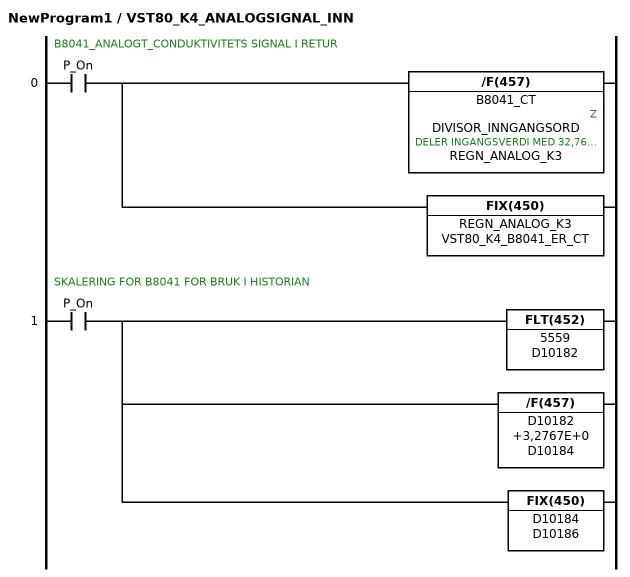
; [picture p480: NewProgram1 / VST80_K4_ANALOGSIGNAL_INN, rungs 0-1]
; rung 0: B8041_ANALOGT_CONDUKTIVITETS SIGNAL I RETUR
LD P_On
/F(457) B8041_CT DIVISOR_INNGANGSORD REGN_ANALOG_K3  ; Z, DELER INGANGSVERDI MED 32,760 FOR OMREGNING TIL 0-1000
FIX(450) REGN_ANALOG_K3 VST80_K4_B8041_ER_CT
; rung 1: SKALERING FOR B8041 FOR BRUK I HISTORIAN
LD P_On
FLT(452) 5559 D10182
/F(457) D10182 +3,2767E+0 D10184
FIX(450) D10184 D10186

### Section VST80_K4_OBJEKTER

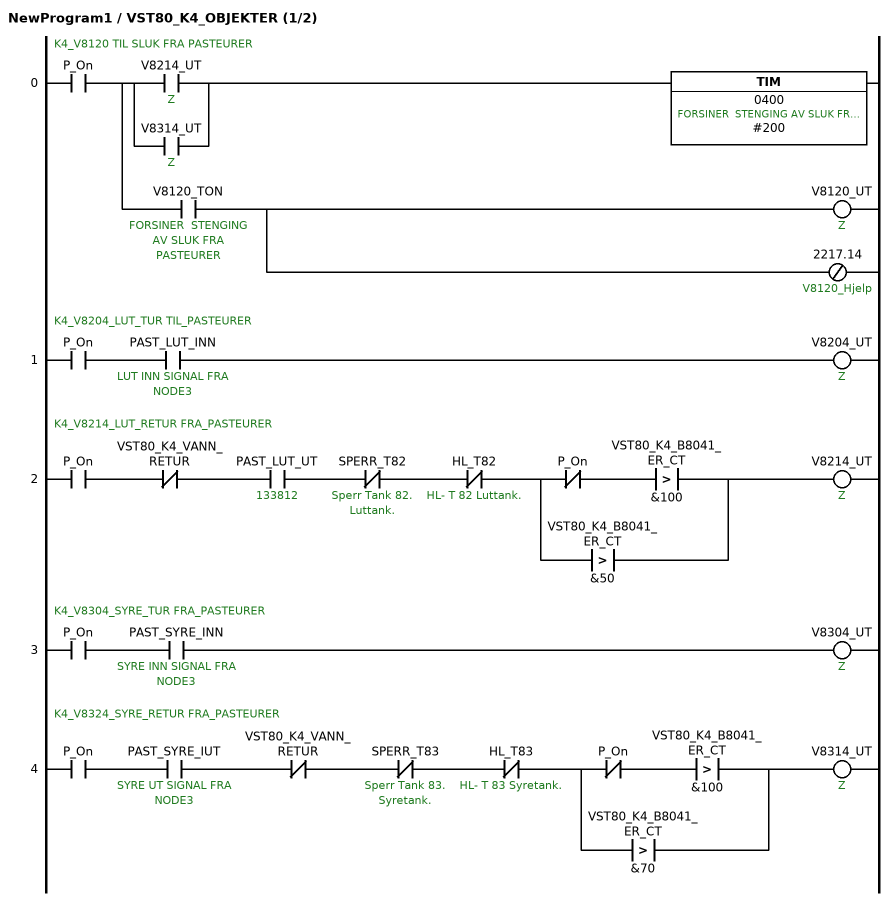
; rung 0: K4_V8120 TIL SLUK FRA PASTEURER
LD P_On
OUT TR0
LD V8214_UT  ; Z
OR V8314_UT  ; Z
ANDLD
TIM 0400 #200  ; FORSINER  STENGING AV SLUK FRA PASTEURER
LD TR0
AND V8120_TON  ; FORSINER  STENGING AV SLUK FRA PASTEURER
OUT V8120_UT  ; Z
OUTNOT 2217.14  ; V8120_Hjelp
; rung 1: K4_V8204_LUT_TUR TIL_PASTEURER
LD P_On
AND PAST_LUT_INN  ; LUT INN SIGNAL FRA NODE3
OUT V8204_UT  ; Z
; rung 2: K4_V8214_LUT_RETUR FRA_PASTEURER
LD P_On
ANDNOT VST80_K4_VANN_RETUR
AND PAST_LUT_UT  ; 133812
ANDNOT SPERR_T82  ; Sperr Tank 82. Luttank.
ANDNOT HL_T82  ; HL- T 82 Luttank.
LDNOT P_On
AND>(320) VST80_K4_B8041_ER_CT &100
OR>(320) VST80_K4_B8041_ER_CT &50
ANDLD
OUT V8214_UT  ; Z
; rung 3: K4_V8304_SYRE_TUR FRA_PASTEURER
LD P_On
AND PAST_SYRE_INN  ; SYRE INN SIGNAL FRA NODE3
OUT V8304_UT  ; Z
; rung 4: K4_V8324_SYRE_RETUR FRA_PASTEURER
LD P_On
AND PAST_SYRE_IUT  ; SYRE UT SIGNAL FRA NODE3
ANDNOT VST80_K4_VANN_RETUR
ANDNOT SPERR_T83  ; Sperr Tank 83. Syretank.
ANDNOT HL_T83  ; HL- T 83 Syretank.
LDNOT P_On
AND>(320) VST80_K4_B8041_ER_CT &100
OR>(320) VST80_K4_B8041_ER_CT &70
ANDLD
OUT V8314_UT  ; Z

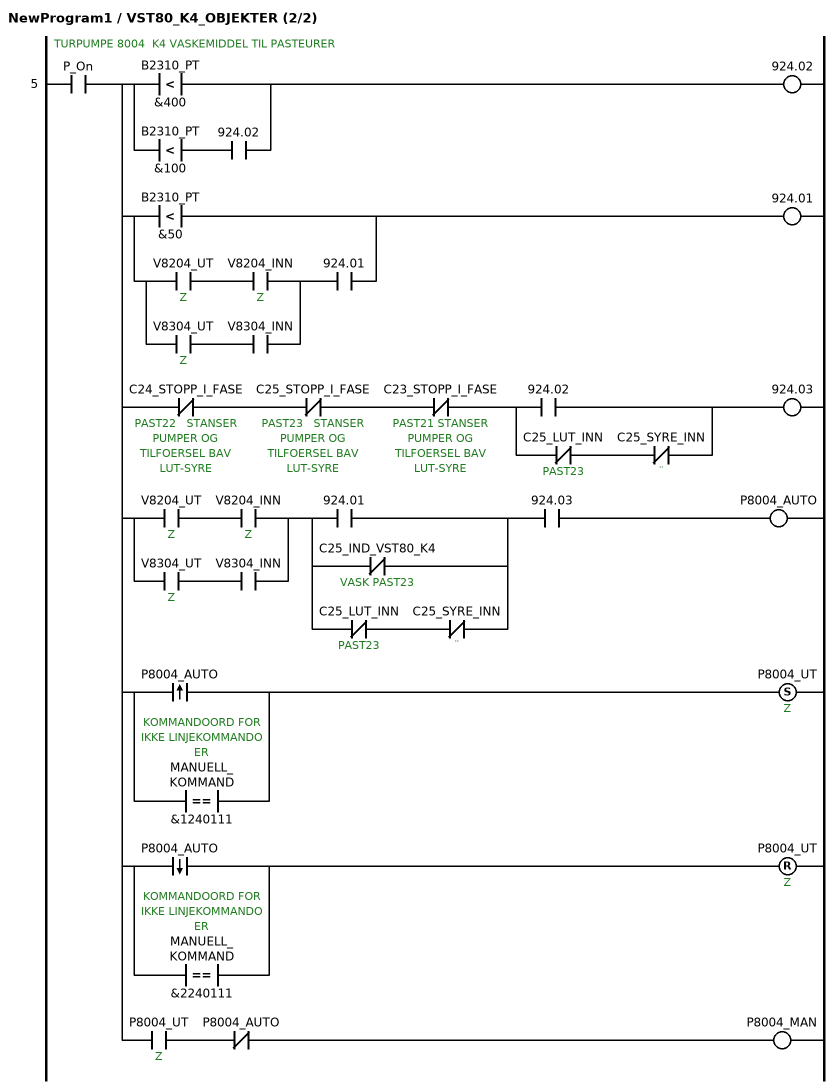
; rung 5: TURPUMPE 8004  K4 VASKEMIDDEL TIL PASTEURER
LD P_On
OUT TR0
LD<(310) B2310_PT &400
LD<(310) B2310_PT &100
AND 924.02
ORLD
ANDLD
OUT 924.02
LD TR0
LD<(310) B2310_PT &50
LD V8204_UT  ; Z
AND V8204_INN  ; Z
LD V8304_UT  ; Z
AND V8304_INN
ORLD
AND 924.01
ORLD
ANDLD
OUT 924.01
LD TR0
ANDNOT C24_STOPP_I_FASE  ; PAST22   STANSER PUMPER OG TILFOERSEL BAV LUT-SYRE
ANDNOT C25_STOPP_I_FASE  ; PAST23   STANSER PUMPER OG TILFOERSEL BAV LUT-SYRE
ANDNOT C23_STOPP_I_FASE  ; PAST21 STANSER PUMPER OG TILFOERSEL BAV LUT-SYRE
LD 924.02
LDNOT C25_LUT_INN  ; PAST23
ANDNOT C25_SYRE_INN  ; ¨
ORLD
ANDLD
OUT 924.03
LD TR0
LD V8204_UT  ; Z
AND V8204_INN  ; Z
LD V8304_UT  ; Z
AND V8304_INN
ORLD
ANDLD
LD 924.01
ORNOT C25_IND_VST80_K4  ; VASK PAST23
LDNOT C25_LUT_INN  ; PAST23
ANDNOT C25_SYRE_INN  ; ¨
ORLD
ANDLD
AND 924.03
OUT P8004_AUTO
LD TR0
@LD P8004_AUTO
OR=L(301) MANUELL_KOMMAND &1240111  ; KOMMANDOORD FOR IKKE LINJEKOMMANDOER
ANDLD
SET P8004_UT  ; Z
LD TR0
%LD P8004_AUTO
OR=L(301) MANUELL_KOMMAND &2240111  ; KOMMANDOORD FOR IKKE LINJEKOMMANDOER
ANDLD
RSET P8004_UT  ; Z
LD TR0
AND P8004_UT  ; Z
ANDNOT P8004_AUTO
OUT P8004_MAN

### Section VST80_FLASH_MOTTAK

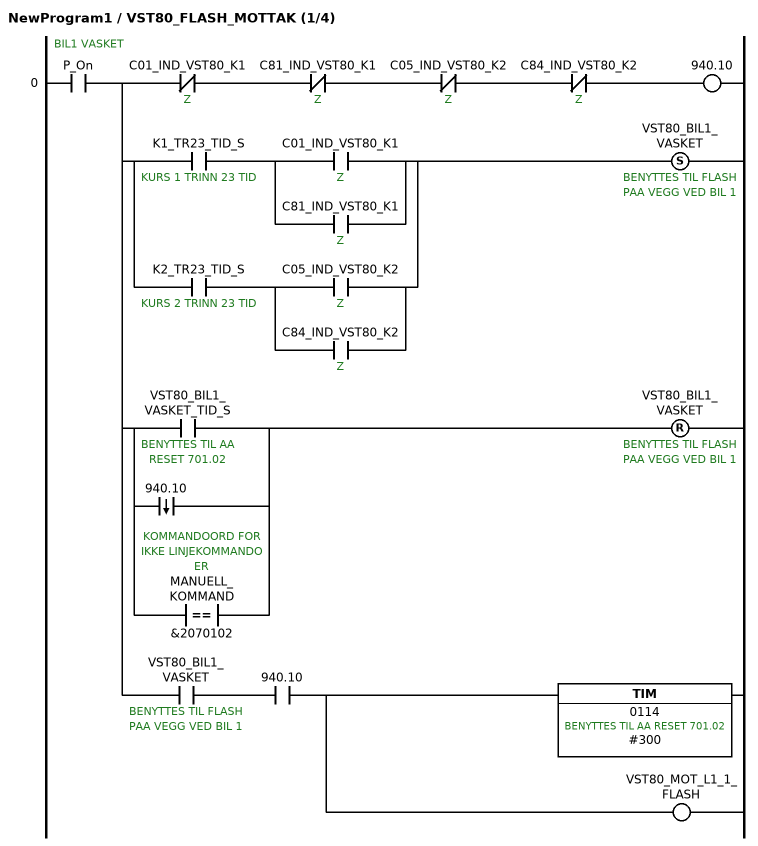
; rung 0: BIL1 VASKET
LD P_On
OUT TR0
ANDNOT C01_IND_VST80_K1  ; Z
ANDNOT C81_IND_VST80_K1  ; Z
ANDNOT C05_IND_VST80_K2  ; Z
ANDNOT C84_IND_VST80_K2  ; Z
OUT 940.10
LD TR0
LD K1_TR23_TID_S  ; KURS 1 TRINN 23 TID
LD C01_IND_VST80_K1  ; Z
OR C81_IND_VST80_K1  ; Z
ANDLD
LD K2_TR23_TID_S  ; KURS 2 TRINN 23 TID
LD C05_IND_VST80_K2  ; Z
OR C84_IND_VST80_K2  ; Z
ANDLD
ORLD
ANDLD
SET VST80_BIL1_VASKET  ; BENYTTES TIL FLASH PAA VEGG VED BIL 1
LD TR0
LD VST80_BIL1_VASKET_TID_S  ; BENYTTES TIL AA RESET 701.02
%OR 940.10
OR=L(301) MANUELL_KOMMAND &2070102  ; KOMMANDOORD FOR IKKE LINJEKOMMANDOER
ANDLD
RSET VST80_BIL1_VASKET  ; BENYTTES TIL FLASH PAA VEGG VED BIL 1
LD TR0
AND VST80_BIL1_VASKET  ; BENYTTES TIL FLASH PAA VEGG VED BIL 1
AND 940.10
TIM 0114 #300  ; BENYTTES TIL AA RESET 701.02
OUT VST80_MOT_L1_1_FLASH

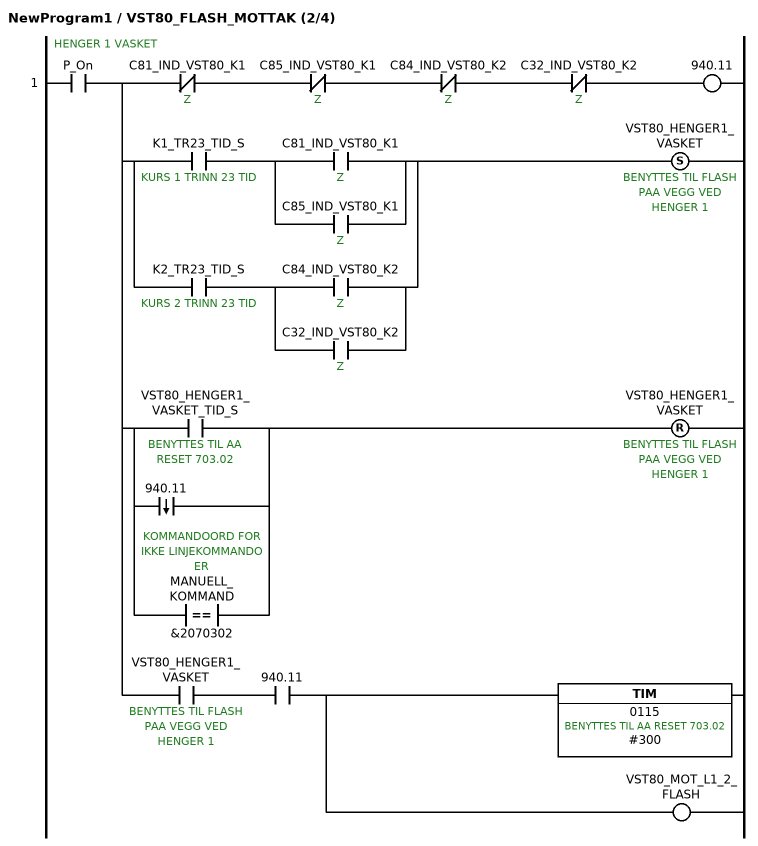
; rung 1: HENGER 1 VASKET
LD P_On
OUT TR0
ANDNOT C81_IND_VST80_K1  ; Z
ANDNOT C85_IND_VST80_K1  ; Z
ANDNOT C84_IND_VST80_K2  ; Z
ANDNOT C32_IND_VST80_K2  ; Z
OUT 940.11
LD TR0
LD K1_TR23_TID_S  ; KURS 1 TRINN 23 TID
LD C81_IND_VST80_K1  ; Z
OR C85_IND_VST80_K1  ; Z
ANDLD
LD K2_TR23_TID_S  ; KURS 2 TRINN 23 TID
LD C84_IND_VST80_K2  ; Z
OR C32_IND_VST80_K2  ; Z
ANDLD
ORLD
ANDLD
SET VST80_HENGER1_VASKET  ; BENYTTES TIL FLASH PAA VEGG VED HENGER 1
LD TR0
LD VST80_HENGER1_VASKET_TID_S  ; BENYTTES TIL AA RESET 703.02
%OR 940.11
OR=L(301) MANUELL_KOMMAND &2070302  ; KOMMANDOORD FOR IKKE LINJEKOMMANDOER
ANDLD
RSET VST80_HENGER1_VASKET  ; BENYTTES TIL FLASH PAA VEGG VED HENGER 1
LD TR0
AND VST80_HENGER1_VASKET  ; BENYTTES TIL FLASH PAA VEGG VED HENGER 1
AND 940.11
TIM 0115 #300  ; BENYTTES TIL AA RESET 703.02
OUT VST80_MOT_L1_2_FLASH

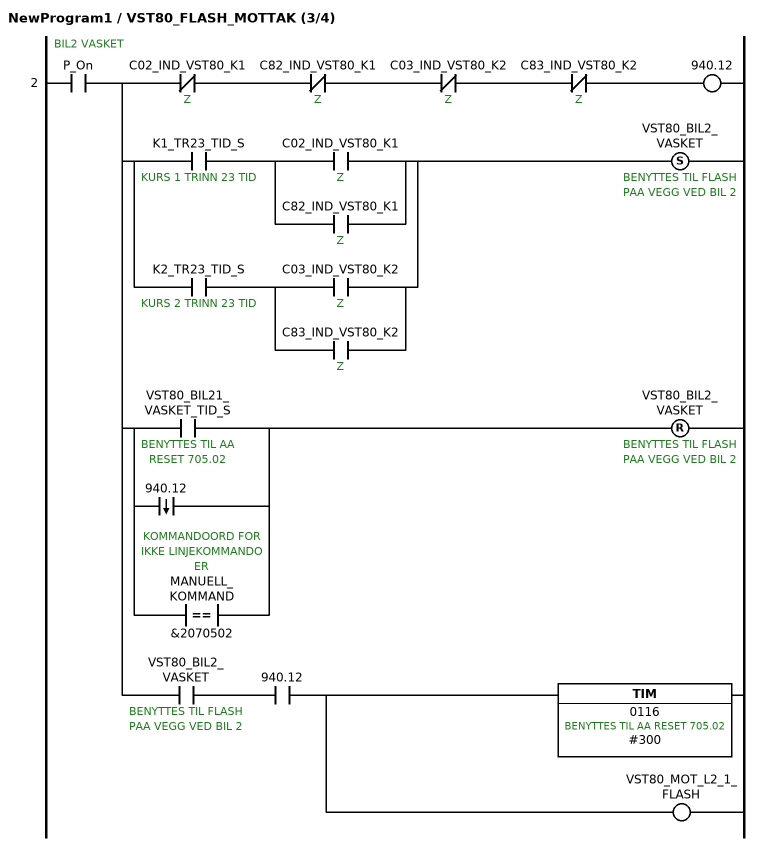
; rung 2: BIL2 VASKET
LD P_On
OUT TR0
ANDNOT C02_IND_VST80_K1  ; Z
ANDNOT C82_IND_VST80_K1  ; Z
ANDNOT C03_IND_VST80_K2  ; Z
ANDNOT C83_IND_VST80_K2  ; Z
OUT 940.12
LD TR0
LD K1_TR23_TID_S  ; KURS 1 TRINN 23 TID
LD C02_IND_VST80_K1  ; Z
OR C82_IND_VST80_K1  ; Z
ANDLD
LD K2_TR23_TID_S  ; KURS 2 TRINN 23 TID
LD C03_IND_VST80_K2  ; Z
OR C83_IND_VST80_K2  ; Z
ANDLD
ORLD
ANDLD
SET VST80_BIL2_VASKET  ; BENYTTES TIL FLASH PAA VEGG VED BIL 2
LD TR0
LD VST80_BIL21_VASKET_TID_S  ; BENYTTES TIL AA RESET 705.02
%OR 940.12
OR=L(301) MANUELL_KOMMAND &2070502  ; KOMMANDOORD FOR IKKE LINJEKOMMANDOER
ANDLD
RSET VST80_BIL2_VASKET  ; BENYTTES TIL FLASH PAA VEGG VED BIL 2
LD TR0
AND VST80_BIL2_VASKET  ; BENYTTES TIL FLASH PAA VEGG VED BIL 2
AND 940.12
TIM 0116 #300  ; BENYTTES TIL AA RESET 705.02
OUT VST80_MOT_L2_1_FLASH

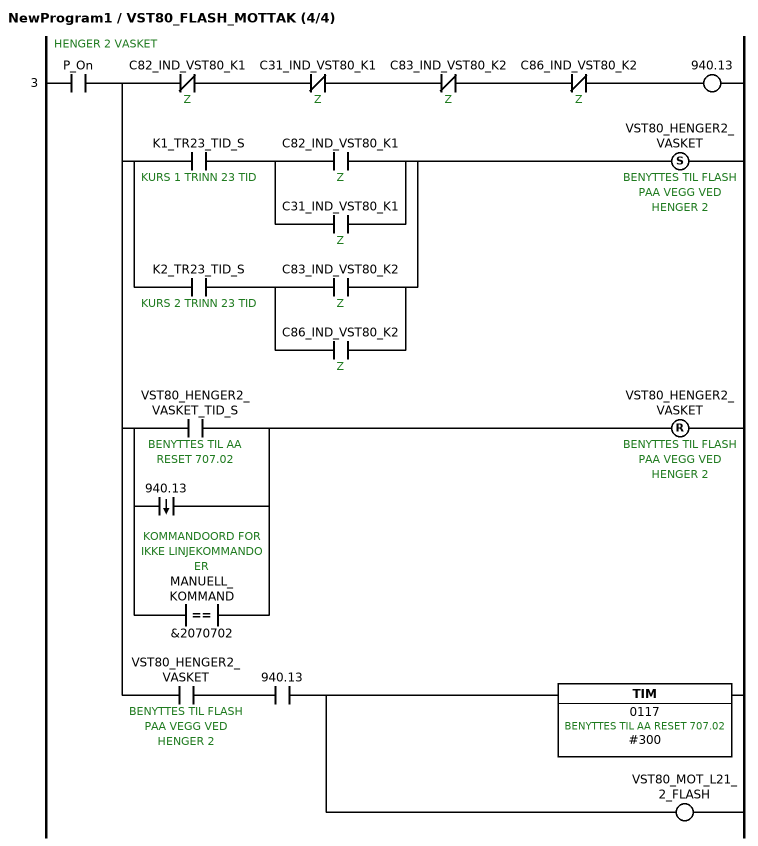
; rung 3: HENGER 2 VASKET
LD P_On
OUT TR0
ANDNOT C82_IND_VST80_K1  ; Z
ANDNOT C31_IND_VST80_K1  ; Z
ANDNOT C83_IND_VST80_K2  ; Z
ANDNOT C86_IND_VST80_K2  ; Z
OUT 940.13
LD TR0
LD K1_TR23_TID_S  ; KURS 1 TRINN 23 TID
LD C82_IND_VST80_K1  ; Z
OR C31_IND_VST80_K1  ; Z
ANDLD
LD K2_TR23_TID_S  ; KURS 2 TRINN 23 TID
LD C83_IND_VST80_K2  ; Z
OR C86_IND_VST80_K2  ; Z
ANDLD
ORLD
ANDLD
SET VST80_HENGER2_VASKET  ; BENYTTES TIL FLASH PAA VEGG VED HENGER 2
LD TR0
LD VST80_HENGER2_VASKET_TID_S  ; BENYTTES TIL AA RESET 707.02
%OR 940.13
OR=L(301) MANUELL_KOMMAND &2070702  ; KOMMANDOORD FOR IKKE LINJEKOMMANDOER
ANDLD
RSET VST80_HENGER2_VASKET  ; BENYTTES TIL FLASH PAA VEGG VED HENGER 2
LD TR0
AND VST80_HENGER2_VASKET  ; BENYTTES TIL FLASH PAA VEGG VED HENGER 2
AND 940.13
TIM 0117 #300  ; BENYTTES TIL AA RESET 707.02
OUT VST80_MOT_L21_2_FLASH

### Section PGM_500_VST80_KURS1

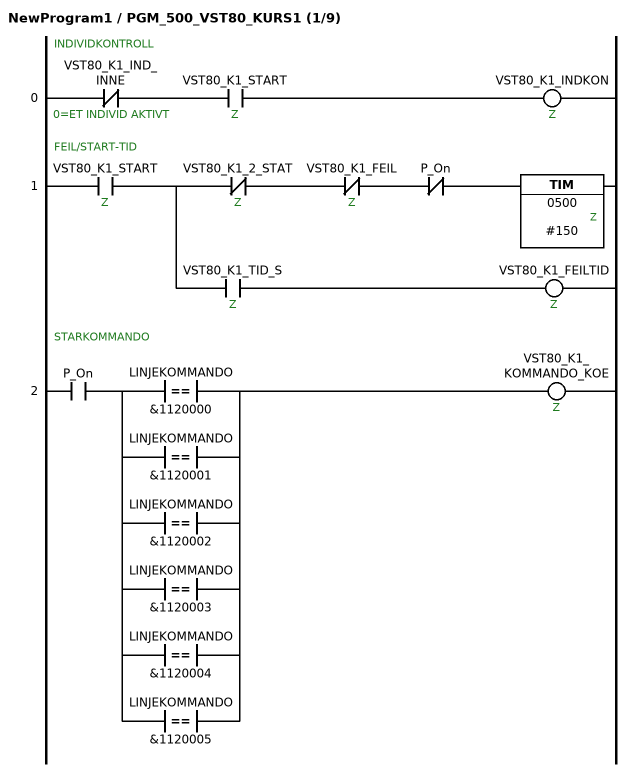
; rung 0: INDIVIDKONTROLL
LDNOT VST80_K1_IND_INNE  ; 0=ET INDIVID AKTIVT
AND VST80_K1_START  ; Z
OUT VST80_K1_INDKON  ; Z
; rung 1: FEIL/START-TID
LD VST80_K1_START  ; Z
OUT TR0
ANDNOT VST80_K1_2_STAT  ; Z
ANDNOT VST80_K1_FEIL  ; Z
ANDNOT P_On
TIM 0500 #150  ; Z
LD TR0
AND VST80_K1_TID_S  ; Z
OUT VST80_K1_FEILTID  ; Z
; rung 2: STARKOMMANDO
LD P_On
LD=L(301) LINJEKOMMANDO &1120000
OR=L(301) LINJEKOMMANDO &1120001
OR=L(301) LINJEKOMMANDO &1120002
OR=L(301) LINJEKOMMANDO &1120003
OR=L(301) LINJEKOMMANDO &1120004
OR=L(301) LINJEKOMMANDO &1120005
ANDLD
OUT VST80_K1_KOMMANDO_KOE  ; Z

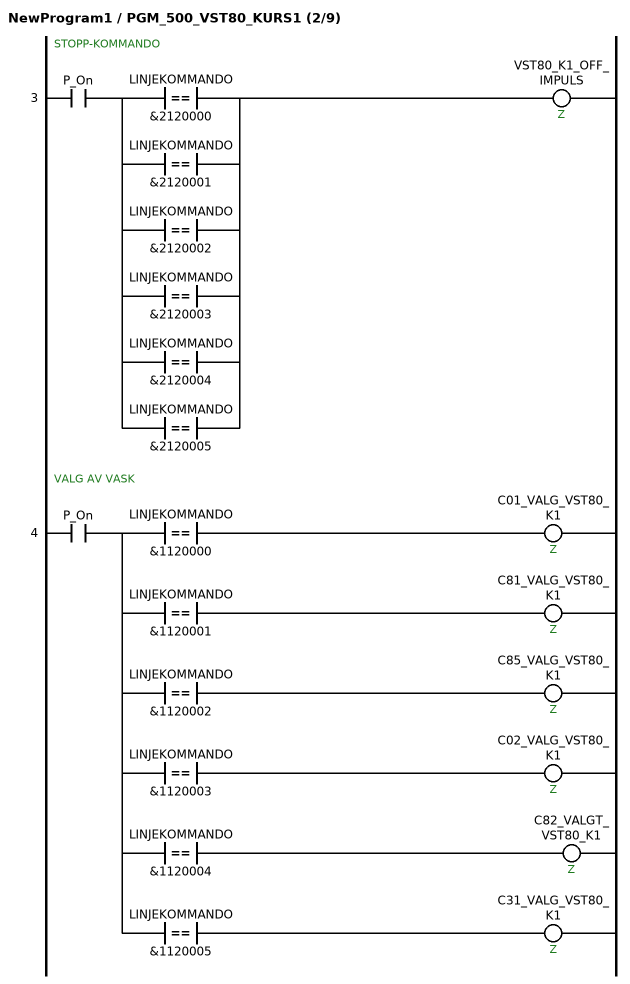
; rung 3: STOPP-KOMMANDO
LD P_On
LD=L(301) LINJEKOMMANDO &2120000
OR=L(301) LINJEKOMMANDO &2120001
OR=L(301) LINJEKOMMANDO &2120002
OR=L(301) LINJEKOMMANDO &2120003
OR=L(301) LINJEKOMMANDO &2120004
OR=L(301) LINJEKOMMANDO &2120005
ANDLD
OUT VST80_K1_OFF_IMPULS  ; Z
; rung 4: VALG AV VASK
LD P_On
OUT TR0
AND=L(301) LINJEKOMMANDO &1120000
OUT C01_VALG_VST80_K1  ; Z
LD TR0
AND=L(301) LINJEKOMMANDO &1120001
OUT C81_VALG_VST80_K1  ; Z
LD TR0
AND=L(301) LINJEKOMMANDO &1120002
OUT C85_VALG_VST80_K1  ; Z
LD TR0
AND=L(301) LINJEKOMMANDO &1120003
OUT C02_VALG_VST80_K1  ; Z
LD TR0
AND=L(301) LINJEKOMMANDO &1120004
OUT C82_VALGT_VST80_K1  ; Z
LD TR0
AND=L(301) LINJEKOMMANDO &1120005
OUT C31_VALG_VST80_K1  ; Z

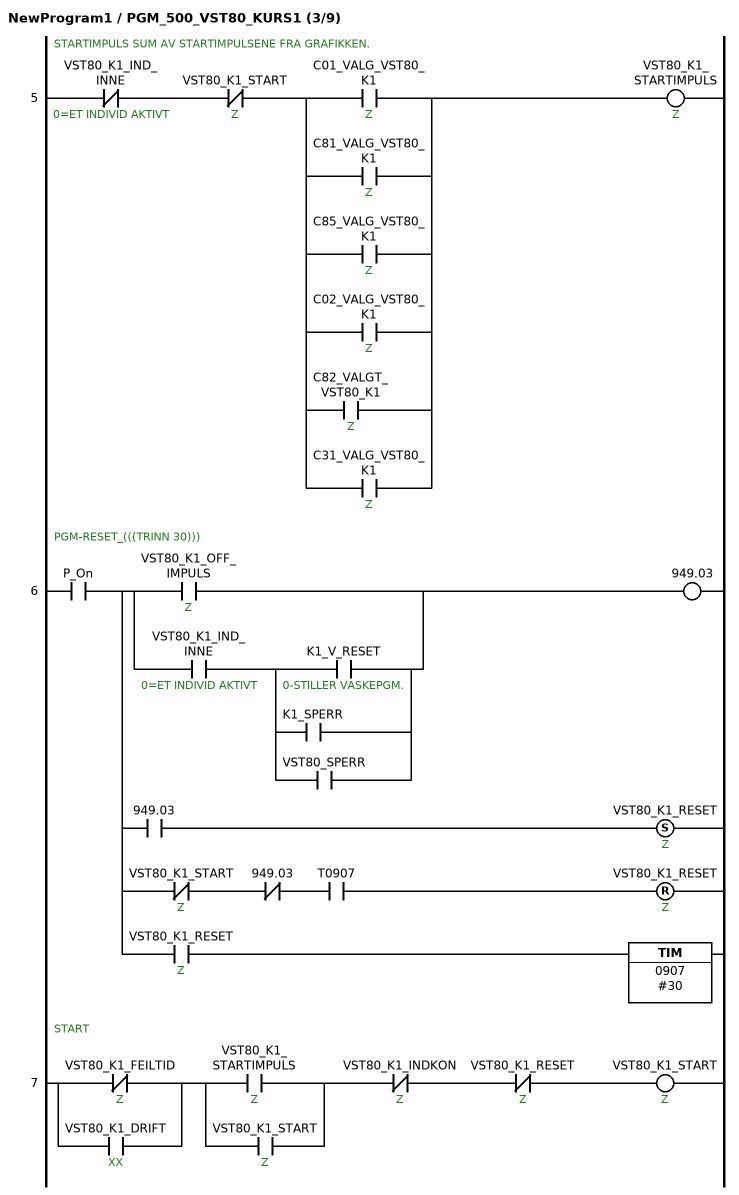
; rung 5: STARTIMPULS SUM AV STARTIMPULSENE FRA GRAFIKKEN.
LDNOT VST80_K1_IND_INNE  ; 0=ET INDIVID AKTIVT
ANDNOT VST80_K1_START  ; Z
LD C01_VALG_VST80_K1  ; Z
OR C81_VALG_VST80_K1  ; Z
OR C85_VALG_VST80_K1  ; Z
OR C02_VALG_VST80_K1  ; Z
OR C82_VALGT_VST80_K1  ; Z
OR C31_VALG_VST80_K1  ; Z
ANDLD
OUT VST80_K1_STARTIMPULS  ; Z
; rung 6: PGM-RESET_(((TRINN 30)))
LD P_On
OUT TR0
LD VST80_K1_OFF_IMPULS  ; Z
LD VST80_K1_IND_INNE  ; 0=ET INDIVID AKTIVT
LD K1_V_RESET  ; 0-STILLER VASKEPGM.
OR K1_SPERR
OR VST80_SPERR
ANDLD
ORLD
ANDLD
OUT 949.03
LD TR0
AND 949.03
SET VST80_K1_RESET  ; Z
LD TR0
ANDNOT VST80_K1_START  ; Z
ANDNOT 949.03
AND T0907
RSET VST80_K1_RESET  ; Z
LD TR0
AND VST80_K1_RESET  ; Z
TIM 0907 #30
; rung 7: START
LDNOT VST80_K1_FEILTID  ; Z
OR VST80_K1_DRIFT  ; XX
LD VST80_K1_STARTIMPULS  ; Z
OR VST80_K1_START  ; Z
ANDLD
ANDNOT VST80_K1_INDKON  ; Z
ANDNOT VST80_K1_RESET  ; Z
OUT VST80_K1_START  ; Z

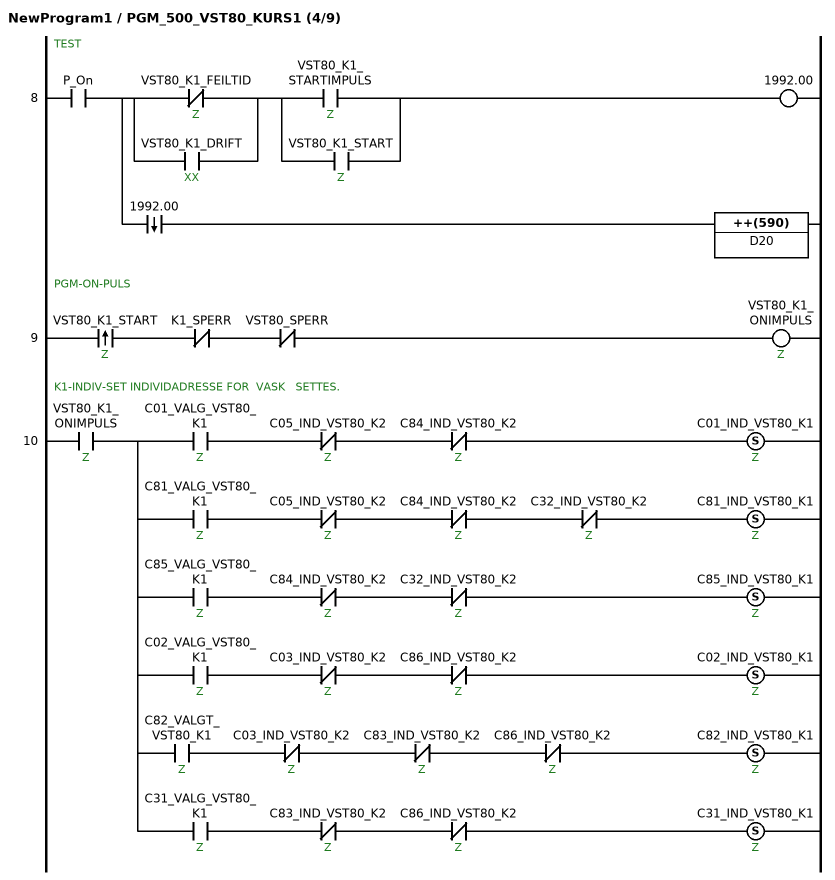
; rung 8: TEST
LD P_On
OUT TR0
LDNOT VST80_K1_FEILTID  ; Z
OR VST80_K1_DRIFT  ; XX
ANDLD
LD VST80_K1_STARTIMPULS  ; Z
OR VST80_K1_START  ; Z
ANDLD
OUT 1992.00
LD TR0
%AND 1992.00
++(590) D20
; rung 9: PGM-ON-PULS
@LD VST80_K1_START  ; Z
ANDNOT K1_SPERR
ANDNOT VST80_SPERR
OUT VST80_K1_ONIMPULS  ; Z
; rung 10: K1-INDIV-SET INDIVIDADRESSE FOR  VASK   SETTES.
LD VST80_K1_ONIMPULS  ; Z
OUT TR0
AND C01_VALG_VST80_K1  ; Z
ANDNOT C05_IND_VST80_K2  ; Z
ANDNOT C84_IND_VST80_K2  ; Z
SET C01_IND_VST80_K1  ; Z
LD TR0
AND C81_VALG_VST80_K1  ; Z
ANDNOT C05_IND_VST80_K2  ; Z
ANDNOT C84_IND_VST80_K2  ; Z
ANDNOT C32_IND_VST80_K2  ; Z
SET C81_IND_VST80_K1  ; Z
LD TR0
AND C85_VALG_VST80_K1  ; Z
ANDNOT C84_IND_VST80_K2  ; Z
ANDNOT C32_IND_VST80_K2  ; Z
SET C85_IND_VST80_K1  ; Z
LD TR0
AND C02_VALG_VST80_K1  ; Z
ANDNOT C03_IND_VST80_K2  ; Z
ANDNOT C86_IND_VST80_K2  ; Z
SET C02_IND_VST80_K1  ; Z
LD TR0
AND C82_VALGT_VST80_K1  ; Z
ANDNOT C03_IND_VST80_K2  ; Z
ANDNOT C83_IND_VST80_K2  ; Z
ANDNOT C86_IND_VST80_K2  ; Z
SET C82_IND_VST80_K1  ; Z
LD TR0
AND C31_VALG_VST80_K1  ; Z
ANDNOT C83_IND_VST80_K2  ; Z
ANDNOT C86_IND_VST80_K2  ; Z
SET C31_IND_VST80_K1  ; Z

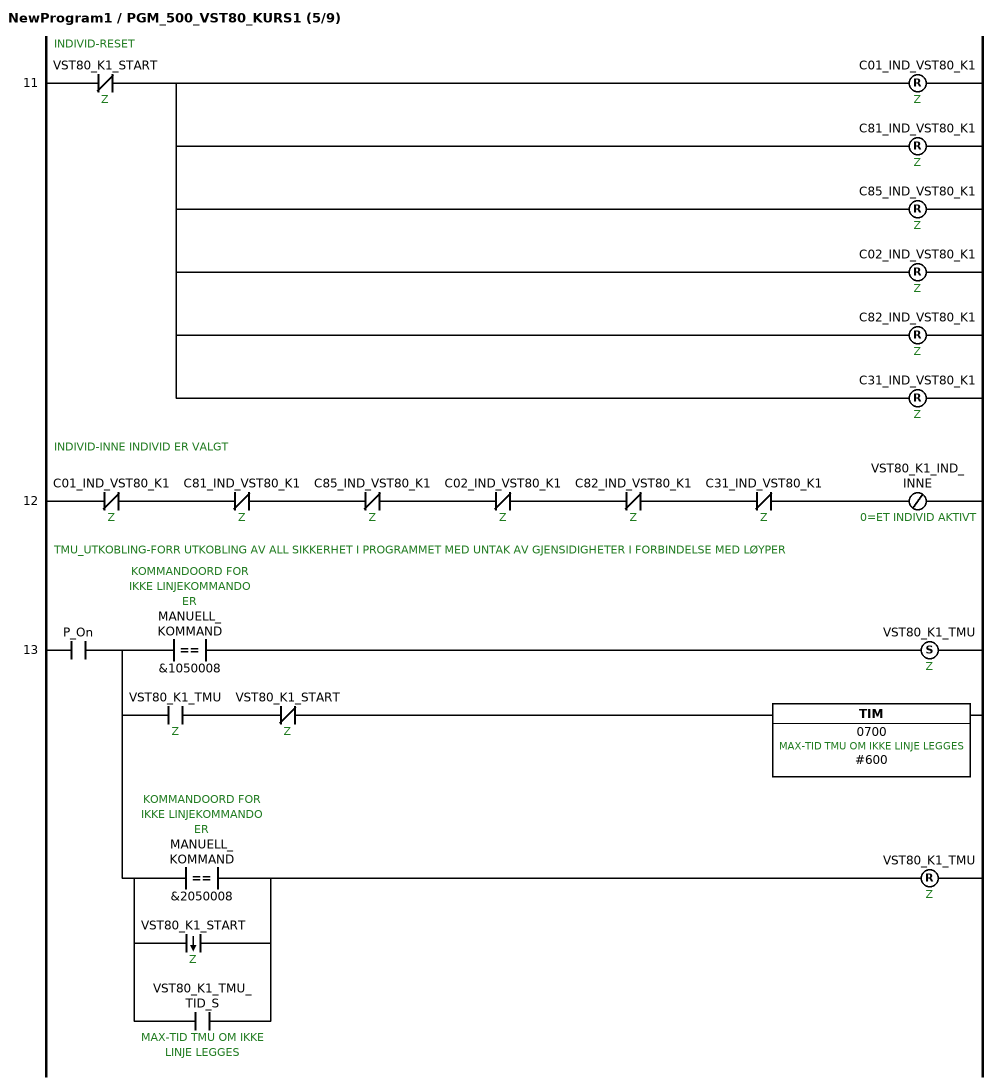
; rung 11: INDIVID-RESET
LDNOT VST80_K1_START  ; Z
RSET C01_IND_VST80_K1  ; Z
RSET C81_IND_VST80_K1  ; Z
RSET C85_IND_VST80_K1  ; Z
RSET C02_IND_VST80_K1  ; Z
RSET C82_IND_VST80_K1  ; Z
RSET C31_IND_VST80_K1  ; Z
; rung 12: INDIVID-INNE INDIVID ER VALGT
LDNOT C01_IND_VST80_K1  ; Z
ANDNOT C81_IND_VST80_K1  ; Z
ANDNOT C85_IND_VST80_K1  ; Z
ANDNOT C02_IND_VST80_K1  ; Z
ANDNOT C82_IND_VST80_K1  ; Z
ANDNOT C31_IND_VST80_K1  ; Z
OUTNOT VST80_K1_IND_INNE  ; 0=ET INDIVID AKTIVT
; rung 13: TMU_UTKOBLING-FORR UTKOBLING AV ALL SIKKERHET I PROGRAMMET MED UNTAK AV GJENSIDIGHETER I FORBINDELSE MED LØYPER
LD P_On
OUT TR0
AND=L(301) MANUELL_KOMMAND &1050008  ; KOMMANDOORD FOR IKKE LINJEKOMMANDOER
SET VST80_K1_TMU  ; Z
LD TR0
AND VST80_K1_TMU  ; Z
ANDNOT VST80_K1_START  ; Z
TIM 0700 #600  ; MAX-TID TMU OM IKKE LINJE LEGGES
LD TR0
LD=L(301) MANUELL_KOMMAND &2050008  ; KOMMANDOORD FOR IKKE LINJEKOMMANDOER
%OR VST80_K1_START  ; Z
OR VST80_K1_TMU_TID_S  ; MAX-TID TMU OM IKKE LINJE LEGGES
ANDLD
RSET VST80_K1_TMU  ; Z

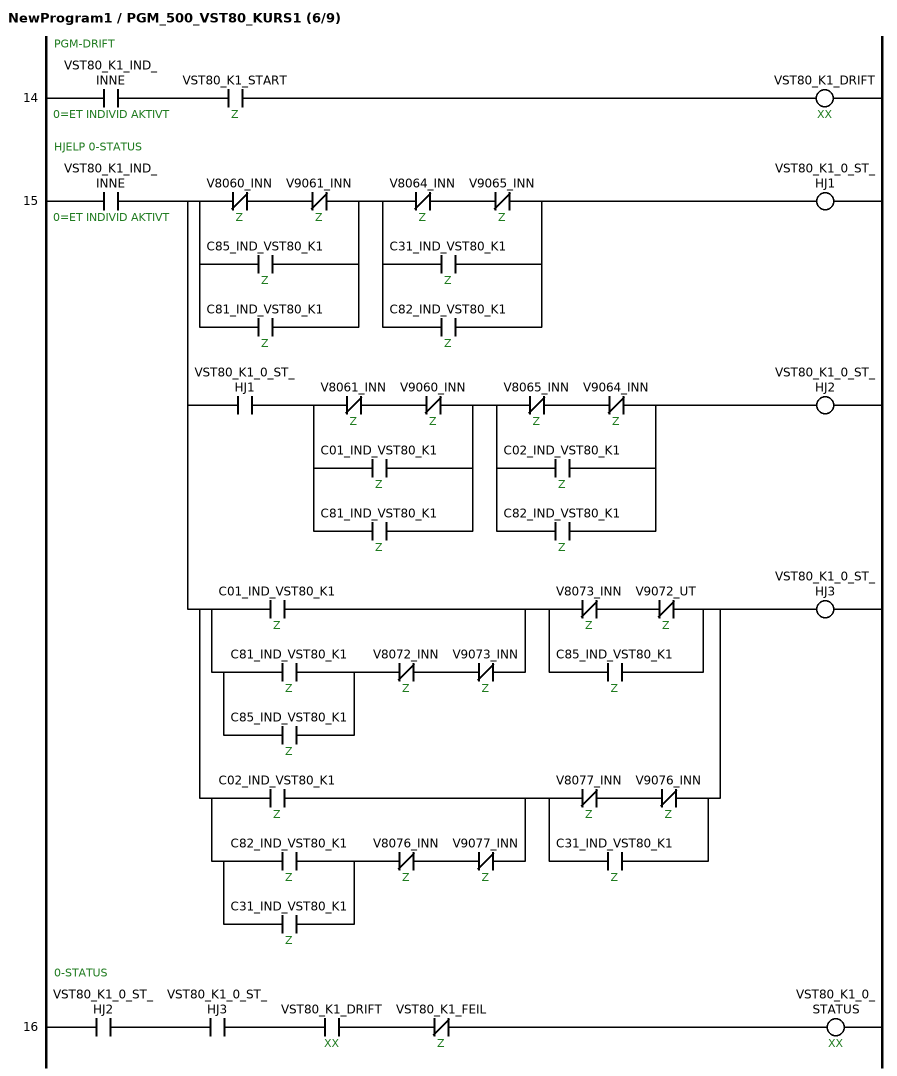
; rung 14: PGM-DRIFT
LD VST80_K1_IND_INNE  ; 0=ET INDIVID AKTIVT
AND VST80_K1_START  ; Z
OUT VST80_K1_DRIFT  ; XX
; rung 15: HJELP 0-STATUS
LD VST80_K1_IND_INNE  ; 0=ET INDIVID AKTIVT
OUT TR0
LDNOT V8060_INN  ; Z
ANDNOT V9061_INN  ; Z
OR C85_IND_VST80_K1  ; Z
OR C81_IND_VST80_K1  ; Z
ANDLD
LDNOT V8064_INN  ; Z
ANDNOT V9065_INN  ; Z
OR C31_IND_VST80_K1  ; Z
OR C82_IND_VST80_K1  ; Z
ANDLD
OUT VST80_K1_0_ST_HJ1
LD TR0
AND VST80_K1_0_ST_HJ1
LDNOT V8061_INN  ; Z
ANDNOT V9060_INN  ; Z
OR C01_IND_VST80_K1  ; Z
OR C81_IND_VST80_K1  ; Z
ANDLD
LDNOT V8065_INN  ; Z
ANDNOT V9064_INN  ; Z
OR C02_IND_VST80_K1  ; Z
OR C82_IND_VST80_K1  ; Z
ANDLD
OUT VST80_K1_0_ST_HJ2
LD TR0
LD C01_IND_VST80_K1  ; Z
LD C81_IND_VST80_K1  ; Z
OR C85_IND_VST80_K1  ; Z
ANDNOT V8072_INN  ; Z
ANDNOT V9073_INN  ; Z
ORLD
LDNOT V8073_INN  ; Z
ANDNOT V9072_UT  ; Z
OR C85_IND_VST80_K1  ; Z
ANDLD
LD C02_IND_VST80_K1  ; Z
LD C82_IND_VST80_K1  ; Z
OR C31_IND_VST80_K1  ; Z
ANDNOT V8076_INN  ; Z
ANDNOT V9077_INN  ; Z
ORLD
LDNOT V8077_INN  ; Z
ANDNOT V9076_INN  ; Z
OR C31_IND_VST80_K1  ; Z
ANDLD
ORLD
ANDLD
OUT VST80_K1_0_ST_HJ3
; rung 16: 0-STATUS
LD VST80_K1_0_ST_HJ2
AND VST80_K1_0_ST_HJ3
AND VST80_K1_DRIFT  ; XX
ANDNOT VST80_K1_FEIL  ; Z
OUT VST80_K1_0_STATUS  ; XX

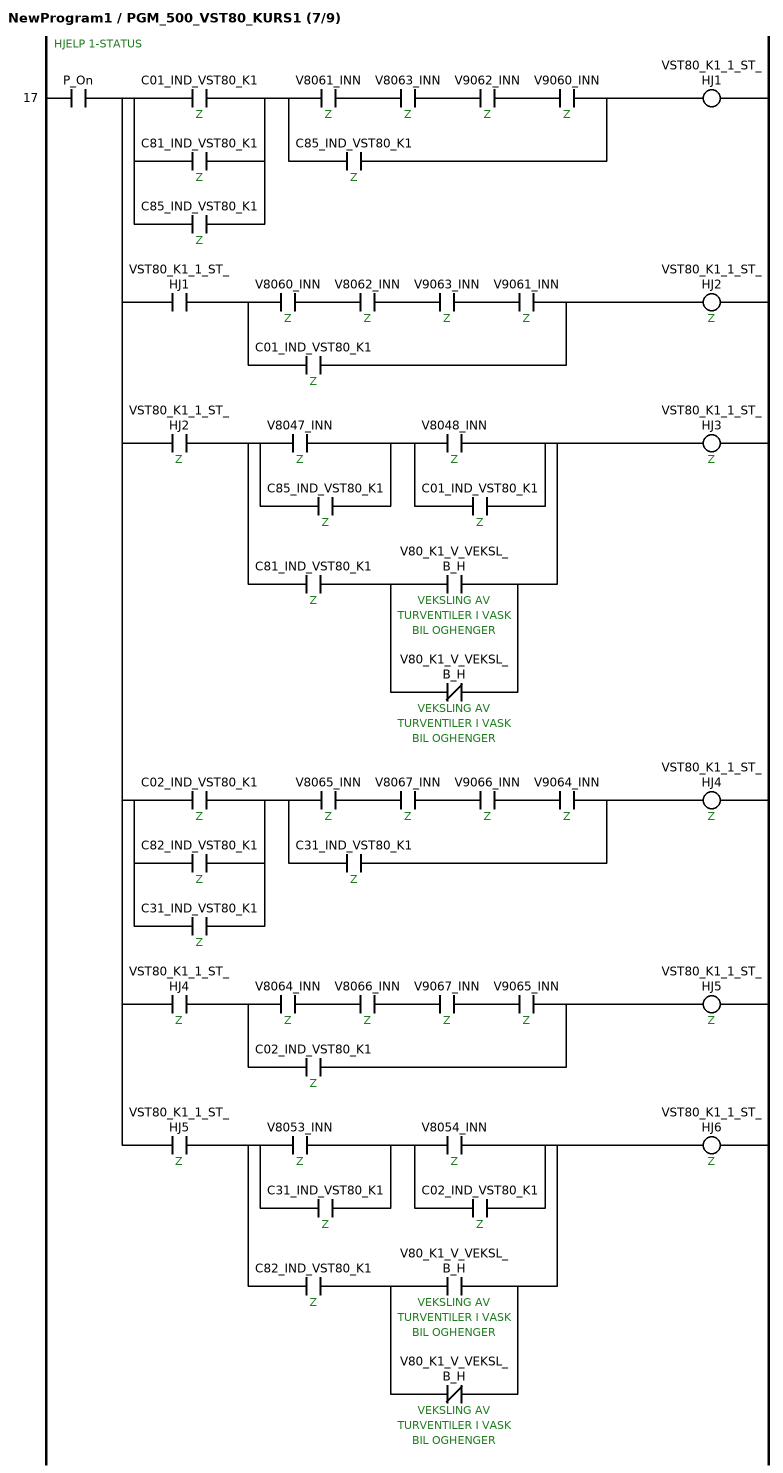
; rung 17: HJELP 1-STATUS
LD P_On
OUT TR0
LD C01_IND_VST80_K1  ; Z
OR C81_IND_VST80_K1  ; Z
OR C85_IND_VST80_K1  ; Z
ANDLD
LD V8061_INN  ; Z
AND V8063_INN  ; Z
AND V9062_INN  ; Z
AND V9060_INN  ; Z
OR C85_IND_VST80_K1  ; Z
ANDLD
OUT VST80_K1_1_ST_HJ1
LD TR0
AND VST80_K1_1_ST_HJ1
LD V8060_INN  ; Z
AND V8062_INN  ; Z
AND V9063_INN  ; Z
AND V9061_INN  ; Z
OR C01_IND_VST80_K1  ; Z
ANDLD
OUT VST80_K1_1_ST_HJ2  ; Z
LD TR0
AND VST80_K1_1_ST_HJ2  ; Z
LD V8047_INN  ; Z
OR C85_IND_VST80_K1  ; Z
LD V8048_INN  ; Z
OR C01_IND_VST80_K1  ; Z
ANDLD
LD C81_IND_VST80_K1  ; Z
LD V80_K1_V_VEKSL_B_H  ; VEKSLING AV TURVENTILER I VASK BIL OGHENGER
ORNOT V80_K1_V_VEKSL_B_H  ; VEKSLING AV TURVENTILER I VASK BIL OGHENGER
ANDLD
ORLD
ANDLD
OUT VST80_K1_1_ST_HJ3  ; Z
LD TR0
LD C02_IND_VST80_K1  ; Z
OR C82_IND_VST80_K1  ; Z
OR C31_IND_VST80_K1  ; Z
ANDLD
LD V8065_INN  ; Z
AND V8067_INN  ; Z
AND V9066_INN  ; Z
AND V9064_INN  ; Z
OR C31_IND_VST80_K1  ; Z
ANDLD
OUT VST80_K1_1_ST_HJ4  ; Z
LD TR0
AND VST80_K1_1_ST_HJ4  ; Z
LD V8064_INN  ; Z
AND V8066_INN  ; Z
AND V9067_INN  ; Z
AND V9065_INN  ; Z
OR C02_IND_VST80_K1  ; Z
ANDLD
OUT VST80_K1_1_ST_HJ5  ; Z
LD TR0
AND VST80_K1_1_ST_HJ5  ; Z
LD V8053_INN  ; Z
OR C31_IND_VST80_K1  ; Z
LD V8054_INN  ; Z
OR C02_IND_VST80_K1  ; Z
ANDLD
LD C82_IND_VST80_K1  ; Z
LD V80_K1_V_VEKSL_B_H  ; VEKSLING AV TURVENTILER I VASK BIL OGHENGER
ORNOT V80_K1_V_VEKSL_B_H  ; VEKSLING AV TURVENTILER I VASK BIL OGHENGER
ANDLD
ORLD
ANDLD
OUT VST80_K1_1_ST_HJ6  ; Z

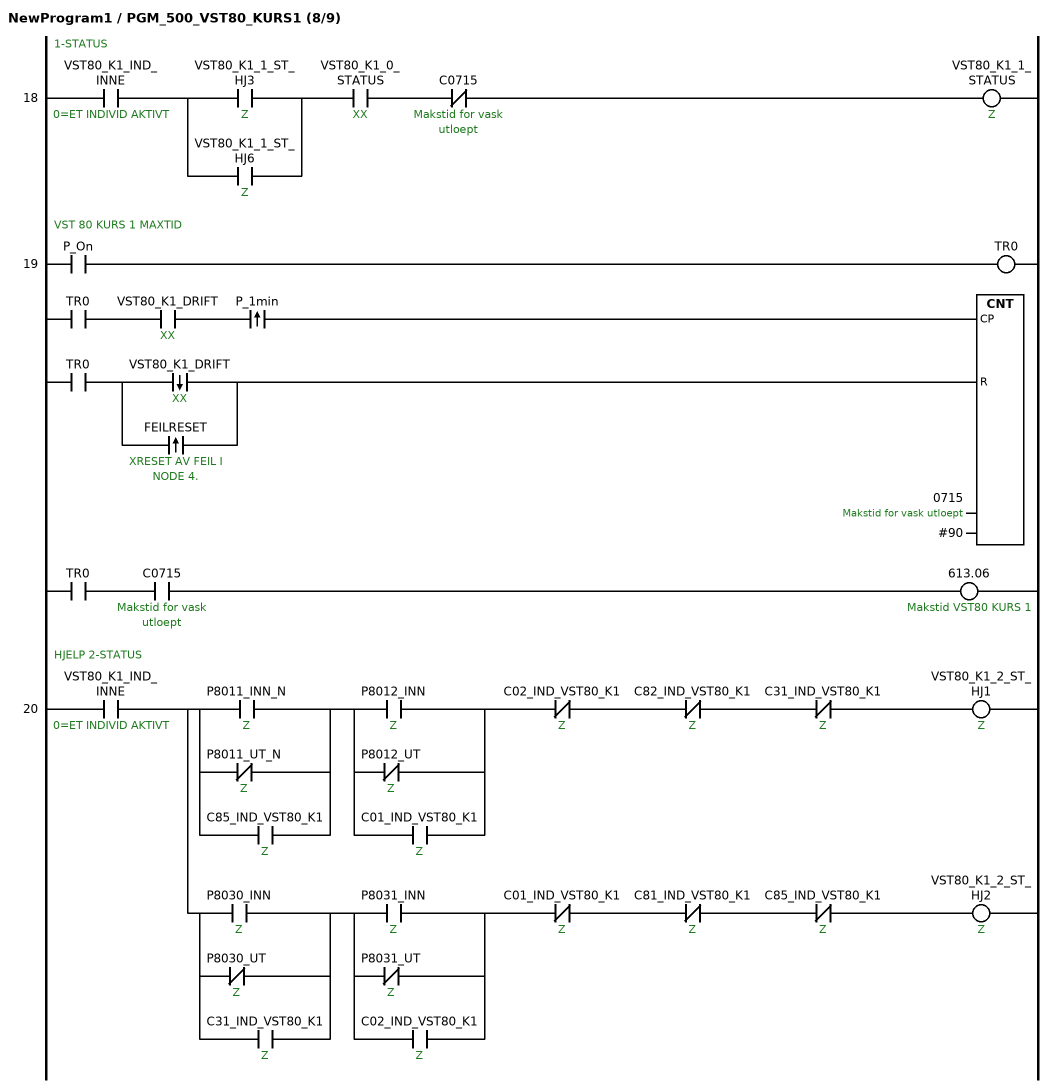
; rung 18: 1-STATUS
LD VST80_K1_IND_INNE  ; 0=ET INDIVID AKTIVT
LD VST80_K1_1_ST_HJ3  ; Z
OR VST80_K1_1_ST_HJ6  ; Z
ANDLD
AND VST80_K1_0_STATUS  ; XX
ANDNOT C0715  ; Makstid for vask utloept
OUT VST80_K1_1_STATUS  ; Z
; rung 19: VST 80 KURS 1 MAXTID
LD P_On
OUT TR0
AND VST80_K1_DRIFT  ; XX
@AND P_1min
LD TR0
%LD VST80_K1_DRIFT  ; XX
@OR FEILRESET  ; XRESET AV FEIL I NODE 4.
ANDLD
CNT 0715 #90  ; Makstid for vask utloept
LD TR0
AND C0715  ; Makstid for vask utloept
OUT 613.06  ; Makstid VST80 KURS 1
; rung 20: HJELP 2-STATUS
LD VST80_K1_IND_INNE  ; 0=ET INDIVID AKTIVT
OUT TR0
LD P8011_INN_N  ; Z
ORNOT P8011_UT_N  ; Z
OR C85_IND_VST80_K1  ; Z
ANDLD
LD P8012_INN  ; Z
ORNOT P8012_UT  ; Z
OR C01_IND_VST80_K1  ; Z
ANDLD
ANDNOT C02_IND_VST80_K1  ; Z
ANDNOT C82_IND_VST80_K1  ; Z
ANDNOT C31_IND_VST80_K1  ; Z
OUT VST80_K1_2_ST_HJ1  ; Z
LD TR0
LD P8030_INN  ; Z
ORNOT P8030_UT  ; Z
OR C31_IND_VST80_K1  ; Z
ANDLD
LD P8031_INN  ; Z
ORNOT P8031_UT  ; Z
OR C02_IND_VST80_K1  ; Z
ANDLD
ANDNOT C01_IND_VST80_K1  ; Z
ANDNOT C81_IND_VST80_K1  ; Z
ANDNOT C85_IND_VST80_K1  ; Z
OUT VST80_K1_2_ST_HJ2  ; Z

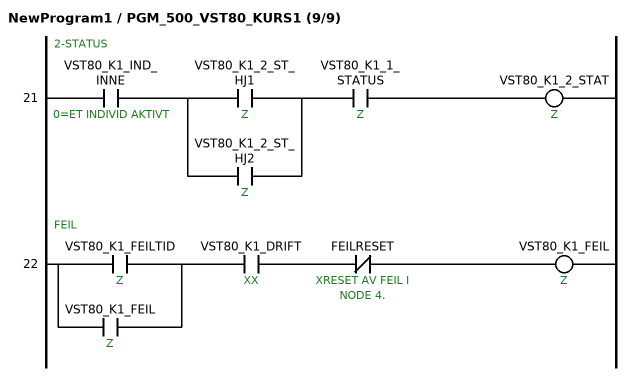
; rung 21: 2-STATUS
LD VST80_K1_IND_INNE  ; 0=ET INDIVID AKTIVT
LD VST80_K1_2_ST_HJ1  ; Z
OR VST80_K1_2_ST_HJ2  ; Z
ANDLD
AND VST80_K1_1_STATUS  ; Z
OUT VST80_K1_2_STAT  ; Z
; rung 22: FEIL
LD VST80_K1_FEILTID  ; Z
OR VST80_K1_FEIL  ; Z
AND VST80_K1_DRIFT  ; XX
ANDNOT FEILRESET  ; XRESET AV FEIL I NODE 4.
OUT VST80_K1_FEIL  ; Z

### Section PGM_501_VST80_KURS2

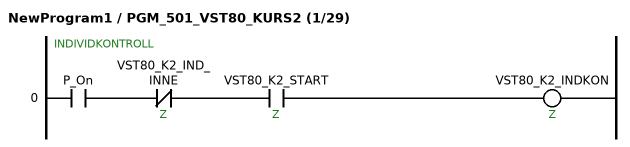
; rung 0: INDIVIDKONTROLL
LD P_On
ANDNOT VST80_K2_IND_INNE  ; Z
AND VST80_K2_START  ; Z
OUT VST80_K2_INDKON  ; Z

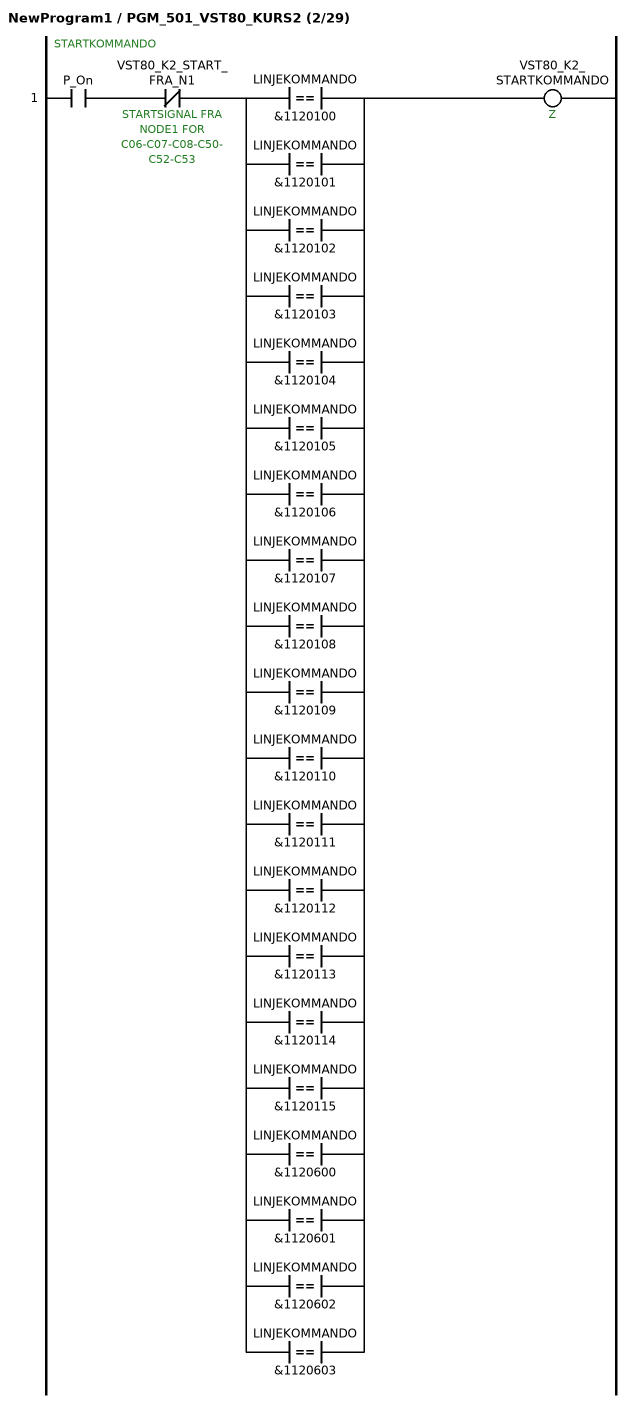
; rung 1: STARTKOMMANDO
LD P_On
ANDNOT VST80_K2_START_FRA_N1  ; STARTSIGNAL FRA NODE1 FOR C06-C07-C08-C50-C52-C53
LD=L(301) LINJEKOMMANDO &1120100
OR=L(301) LINJEKOMMANDO &1120101
OR=L(301) LINJEKOMMANDO &1120102
OR=L(301) LINJEKOMMANDO &1120103
OR=L(301) LINJEKOMMANDO &1120104
OR=L(301) LINJEKOMMANDO &1120105
OR=L(301) LINJEKOMMANDO &1120106
OR=L(301) LINJEKOMMANDO &1120107
OR=L(301) LINJEKOMMANDO &1120108
OR=L(301) LINJEKOMMANDO &1120109
OR=L(301) LINJEKOMMANDO &1120110
OR=L(301) LINJEKOMMANDO &1120111
OR=L(301) LINJEKOMMANDO &1120112
OR=L(301) LINJEKOMMANDO &1120113
OR=L(301) LINJEKOMMANDO &1120114
OR=L(301) LINJEKOMMANDO &1120115
OR=L(301) LINJEKOMMANDO &1120600
OR=L(301) LINJEKOMMANDO &1120601
OR=L(301) LINJEKOMMANDO &1120602
OR=L(301) LINJEKOMMANDO &1120603
ANDLD
OUT VST80_K2_STARTKOMMANDO  ; Z

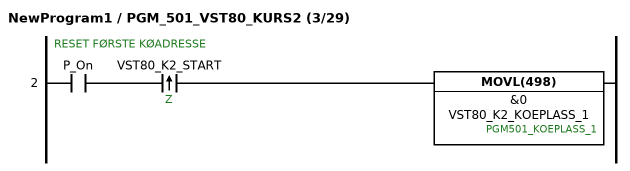
; rung 2: RESET FØRSTE KØADRESSE
LD P_On
@AND VST80_K2_START  ; Z
MOVL(498) &0 VST80_K2_KOEPLASS_1  ; PGM501_KOEPLASS_1

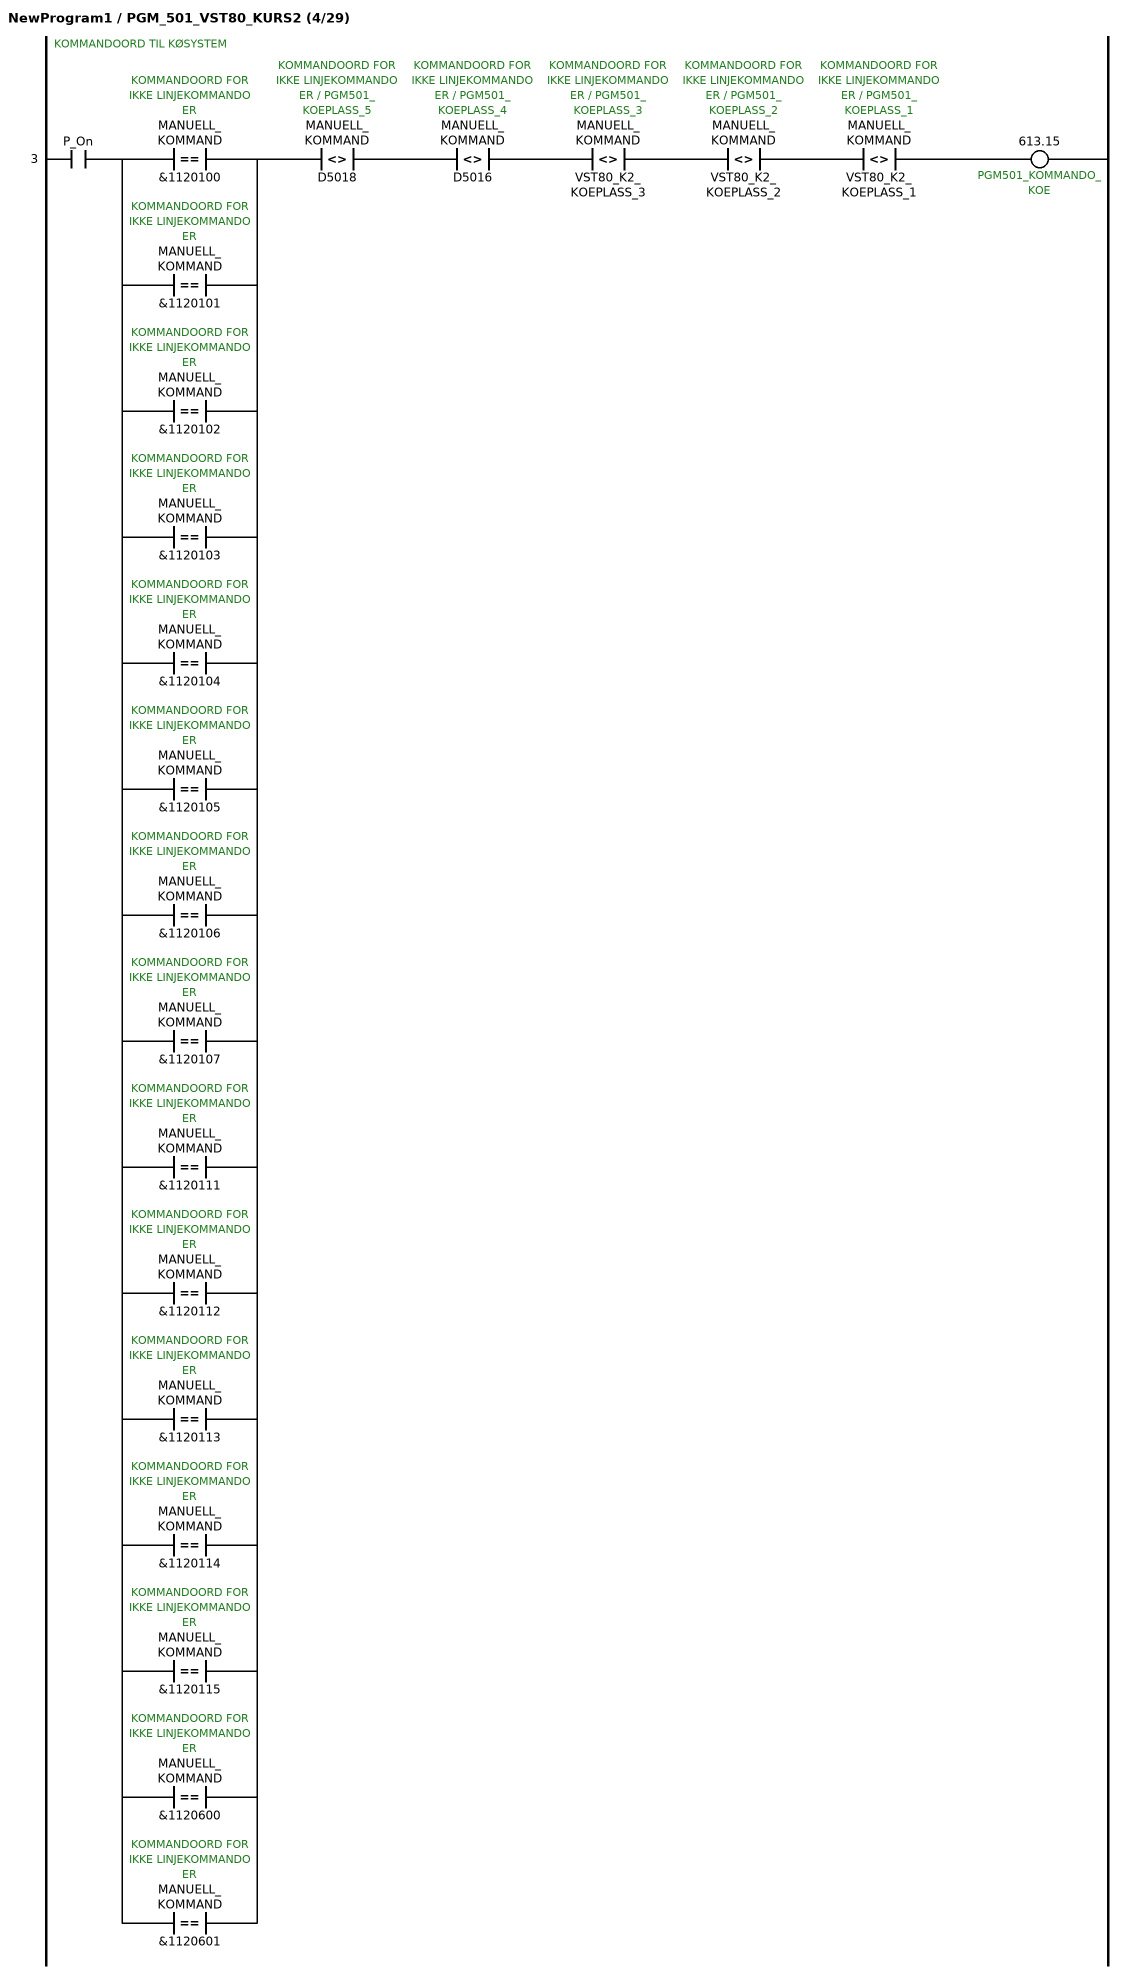
; rung 3: KOMMANDOORD TIL KØSYSTEM
LD P_On
LD=L(301) MANUELL_KOMMAND &1120100  ; KOMMANDOORD FOR IKKE LINJEKOMMANDOER
OR=L(301) MANUELL_KOMMAND &1120101  ; KOMMANDOORD FOR IKKE LINJEKOMMANDOER
OR=L(301) MANUELL_KOMMAND &1120102  ; KOMMANDOORD FOR IKKE LINJEKOMMANDOER
OR=L(301) MANUELL_KOMMAND &1120103  ; KOMMANDOORD FOR IKKE LINJEKOMMANDOER
OR=L(301) MANUELL_KOMMAND &1120104  ; KOMMANDOORD FOR IKKE LINJEKOMMANDOER
OR=L(301) MANUELL_KOMMAND &1120105  ; KOMMANDOORD FOR IKKE LINJEKOMMANDOER
OR=L(301) MANUELL_KOMMAND &1120106  ; KOMMANDOORD FOR IKKE LINJEKOMMANDOER
OR=L(301) MANUELL_KOMMAND &1120107  ; KOMMANDOORD FOR IKKE LINJEKOMMANDOER
OR=L(301) MANUELL_KOMMAND &1120111  ; KOMMANDOORD FOR IKKE LINJEKOMMANDOER
OR=L(301) MANUELL_KOMMAND &1120112  ; KOMMANDOORD FOR IKKE LINJEKOMMANDOER
OR=L(301) MANUELL_KOMMAND &1120113  ; KOMMANDOORD FOR IKKE LINJEKOMMANDOER
OR=L(301) MANUELL_KOMMAND &1120114  ; KOMMANDOORD FOR IKKE LINJEKOMMANDOER
OR=L(301) MANUELL_KOMMAND &1120115  ; KOMMANDOORD FOR IKKE LINJEKOMMANDOER
OR=L(301) MANUELL_KOMMAND &1120600  ; KOMMANDOORD FOR IKKE LINJEKOMMANDOER
OR=L(301) MANUELL_KOMMAND &1120601  ; KOMMANDOORD FOR IKKE LINJEKOMMANDOER
ANDLD
AND<>L(306) MANUELL_KOMMAND D5018  ; KOMMANDOORD FOR IKKE LINJEKOMMANDOER, PGM501_KOEPLASS_5
AND<>L(306) MANUELL_KOMMAND D5016  ; KOMMANDOORD FOR IKKE LINJEKOMMANDOER, PGM501_KOEPLASS_4
AND<>L(306) MANUELL_KOMMAND VST80_K2_KOEPLASS_3  ; KOMMANDOORD FOR IKKE LINJEKOMMANDOER, PGM501_KOEPLASS_3
AND<>L(306) MANUELL_KOMMAND VST80_K2_KOEPLASS_2  ; KOMMANDOORD FOR IKKE LINJEKOMMANDOER, PGM501_KOEPLASS_2
AND<>L(306) MANUELL_KOMMAND VST80_K2_KOEPLASS_1  ; KOMMANDOORD FOR IKKE LINJEKOMMANDOER, PGM501_KOEPLASS_1
OUT 613.15  ; PGM501_KOMMANDO_KOE

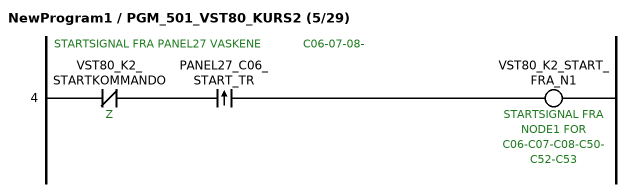
; rung 4: STARTSIGNAL FRA PANEL27 VASKENE            C06-07-08-
LDNOT VST80_K2_STARTKOMMANDO  ; Z
@AND PANEL27_C06_START_TR
OUT VST80_K2_START_FRA_N1  ; STARTSIGNAL FRA NODE1 FOR C06-C07-C08-C50-C52-C53

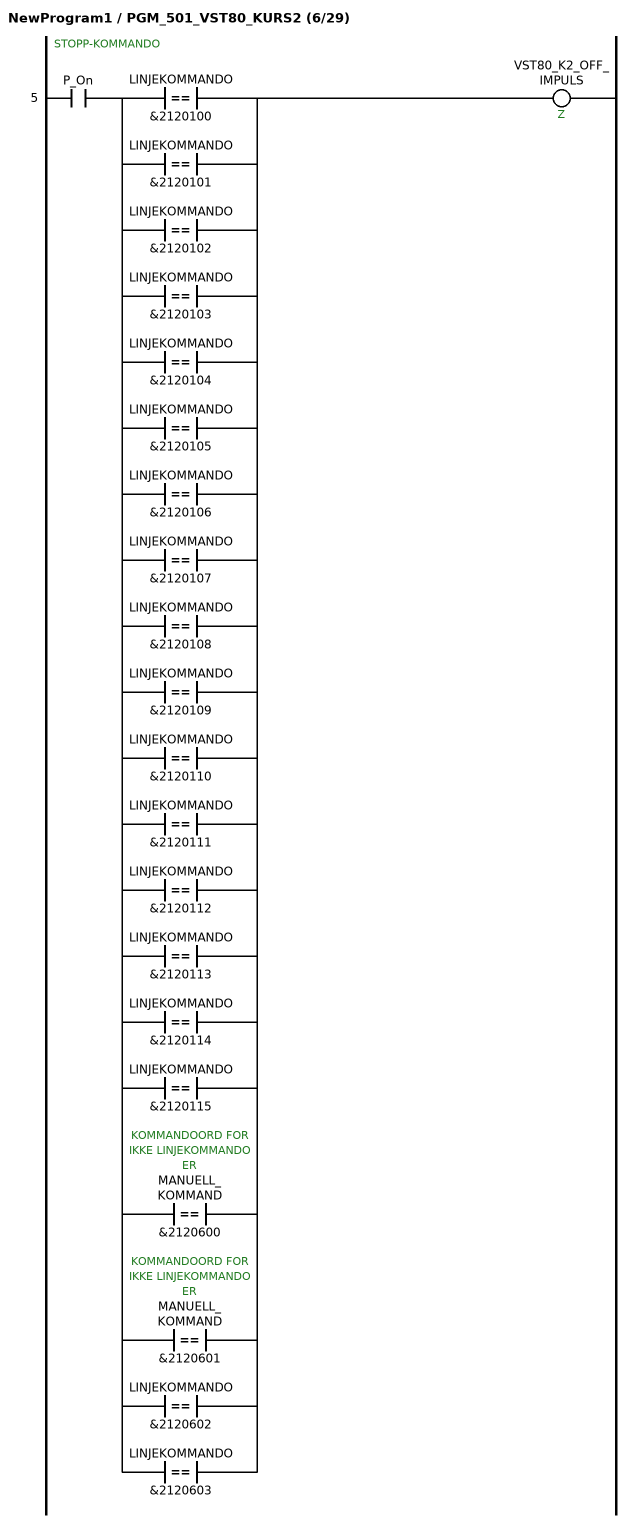
; rung 5: STOPP-KOMMANDO
LD P_On
LD=L(301) LINJEKOMMANDO &2120100
OR=L(301) LINJEKOMMANDO &2120101
OR=L(301) LINJEKOMMANDO &2120102
OR=L(301) LINJEKOMMANDO &2120103
OR=L(301) LINJEKOMMANDO &2120104
OR=L(301) LINJEKOMMANDO &2120105
OR=L(301) LINJEKOMMANDO &2120106
OR=L(301) LINJEKOMMANDO &2120107
OR=L(301) LINJEKOMMANDO &2120108
OR=L(301) LINJEKOMMANDO &2120109
OR=L(301) LINJEKOMMANDO &2120110
OR=L(301) LINJEKOMMANDO &2120111
OR=L(301) LINJEKOMMANDO &2120112
OR=L(301) LINJEKOMMANDO &2120113
OR=L(301) LINJEKOMMANDO &2120114
OR=L(301) LINJEKOMMANDO &2120115
OR=L(301) MANUELL_KOMMAND &2120600  ; KOMMANDOORD FOR IKKE LINJEKOMMANDOER
OR=L(301) MANUELL_KOMMAND &2120601  ; KOMMANDOORD FOR IKKE LINJEKOMMANDOER
OR=L(301) LINJEKOMMANDO &2120602
OR=L(301) LINJEKOMMANDO &2120603
ANDLD
OUT VST80_K2_OFF_IMPULS  ; Z

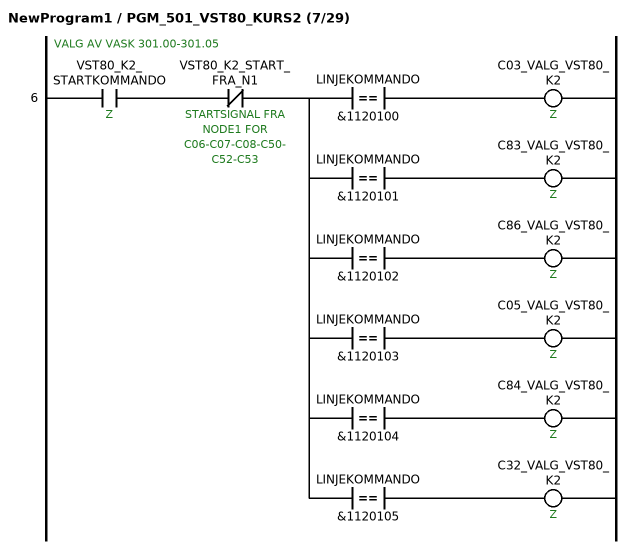
; rung 6: VALG AV VASK 301.00-301.05
LD VST80_K2_STARTKOMMANDO  ; Z
ANDNOT VST80_K2_START_FRA_N1  ; STARTSIGNAL FRA NODE1 FOR C06-C07-C08-C50-C52-C53
OUT TR0
AND=L(301) LINJEKOMMANDO &1120100
OUT C03_VALG_VST80_K2  ; Z
LD TR0
AND=L(301) LINJEKOMMANDO &1120101
OUT C83_VALG_VST80_K2  ; Z
LD TR0
AND=L(301) LINJEKOMMANDO &1120102
OUT C86_VALG_VST80_K2  ; Z
LD TR0
AND=L(301) LINJEKOMMANDO &1120103
OUT C05_VALG_VST80_K2  ; Z
LD TR0
AND=L(301) LINJEKOMMANDO &1120104
OUT C84_VALG_VST80_K2  ; Z
LD TR0
AND=L(301) LINJEKOMMANDO &1120105
OUT C32_VALG_VST80_K2  ; Z

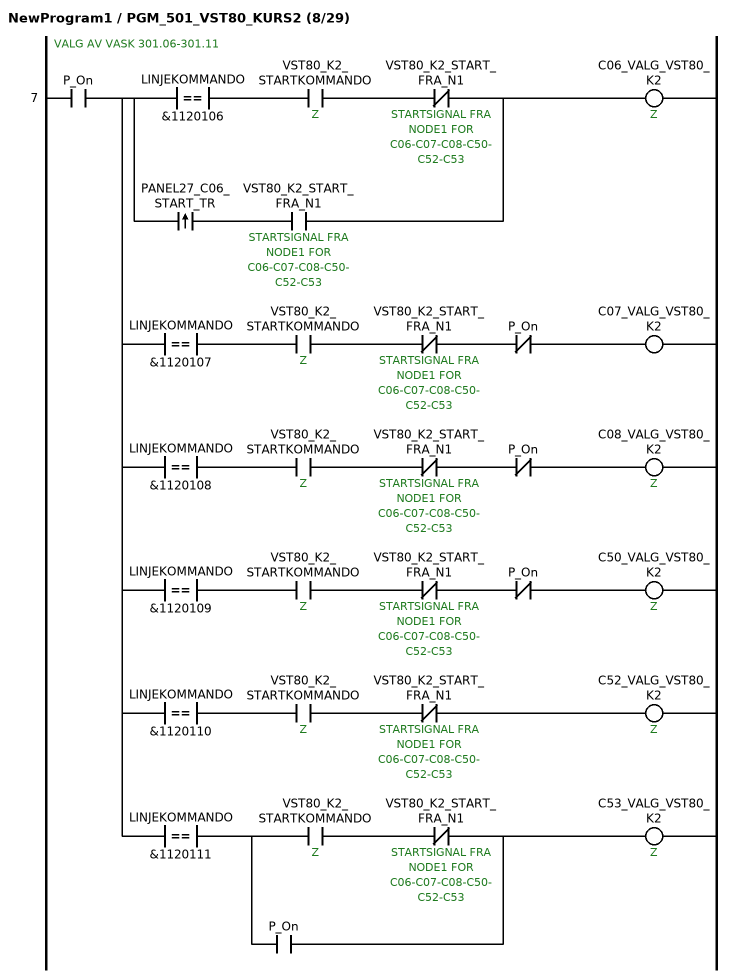
; rung 7: VALG AV VASK 301.06-301.11
LD P_On
OUT TR0
LD=L(301) LINJEKOMMANDO &1120106
AND VST80_K2_STARTKOMMANDO  ; Z
ANDNOT VST80_K2_START_FRA_N1  ; STARTSIGNAL FRA NODE1 FOR C06-C07-C08-C50-C52-C53
@LD PANEL27_C06_START_TR
AND VST80_K2_START_FRA_N1  ; STARTSIGNAL FRA NODE1 FOR C06-C07-C08-C50-C52-C53
ORLD
ANDLD
OUT C06_VALG_VST80_K2  ; Z
LD TR0
AND=L(301) LINJEKOMMANDO &1120107
AND VST80_K2_STARTKOMMANDO  ; Z
ANDNOT VST80_K2_START_FRA_N1  ; STARTSIGNAL FRA NODE1 FOR C06-C07-C08-C50-C52-C53
ANDNOT P_On
OUT C07_VALG_VST80_K2
LD TR0
AND=L(301) LINJEKOMMANDO &1120108
AND VST80_K2_STARTKOMMANDO  ; Z
ANDNOT VST80_K2_START_FRA_N1  ; STARTSIGNAL FRA NODE1 FOR C06-C07-C08-C50-C52-C53
ANDNOT P_On
OUT C08_VALG_VST80_K2  ; Z
LD TR0
AND=L(301) LINJEKOMMANDO &1120109
AND VST80_K2_STARTKOMMANDO  ; Z
ANDNOT VST80_K2_START_FRA_N1  ; STARTSIGNAL FRA NODE1 FOR C06-C07-C08-C50-C52-C53
ANDNOT P_On
OUT C50_VALG_VST80_K2  ; Z
LD TR0
AND=L(301) LINJEKOMMANDO &1120110
AND VST80_K2_STARTKOMMANDO  ; Z
ANDNOT VST80_K2_START_FRA_N1  ; STARTSIGNAL FRA NODE1 FOR C06-C07-C08-C50-C52-C53
OUT C52_VALG_VST80_K2  ; Z
LD TR0
AND=L(301) LINJEKOMMANDO &1120111
LD VST80_K2_STARTKOMMANDO  ; Z
ANDNOT VST80_K2_START_FRA_N1  ; STARTSIGNAL FRA NODE1 FOR C06-C07-C08-C50-C52-C53
OR P_On
ANDLD
OUT C53_VALG_VST80_K2  ; Z

